PROGRAM MAIN
VAR
	

END_VAR

{IF hasattribute (GVL_RealTimeLogging,'enabled')}
	// if you add the TC3_RealtimeMonitoring library then the project will automatically switch to Performance test. 
	PerformanceTest();
{ELSE}
	ExampleApplication();
{END_IF}

END_PROGRAM

(* stored: Version 1.1.0.1, ProductVersion 3.1.4024.5
   POU MAIN: Id {b0e54dca-c4a4-474e-8a8e-b46682f13b27}, SpecialFunc None *)
